# EPICS substitutions: nfsDir/asExample/db/user.substitutions
# Example substitutions file

file "db/dbExample1.db" {
    { user = "long" }
}

file db/dbExample2.db {
    pattern { user, no, scan }
        { "long", 1, "1 second" }
        { "long", 2, "2 second" }
        { "long", 3, "5 second" }
}
